# EPICS substitutions: viocs/si_ps/si_psApp/Db/sdb0.substitutions
file "db/individual.db" {
    pattern { family, pos, num }
        { "SDB0", "02M1", "" }
        { "SDB0", "02M2", "" }
        { "SDB0", "04M1", "" }
        { "SDB0", "04M2", "" }
        { "SDB0", "06M1", "" }
        { "SDB0", "06M2", "" }
        { "SDB0", "08M1", "" }
        { "SDB0", "08M2", "" }
        { "SDB0", "10M1", "" }
        { "SDB0", "10M2", "" }
        { "SDB0", "12M1", "" }
        { "SDB0", "12M2", "" }
        { "SDB0", "14M1", "" }
        { "SDB0", "14M2", "" }
        { "SDB0", "16M1", "" }
        { "SDB0", "16M2", "" }
        { "SDB0", "18M1", "" }
        { "SDB0", "18M2", "" }
        { "SDB0", "20M1", "" }
        { "SDB0", "20M2", "" }
}
